(* IEC 61131-3 sources: RL_MAR/experiments/comparison/autoplc/results/deepseek-ai-DeepSeek-V3.2_20260508_111905/med_63, 1 file *)

(* ---- med_63_3.st ---- *)
FUNCTION MoveCarToExitGate : BOOL
VAR_INPUT
    SpaceNumber : INT;
END_VAR
VAR
    // Local variables if needed
END_VAR

(* This function simulates car movement to exit gate *)
(* In a real implementation, this would control physical actuators *)
(* For this example, we'll return TRUE immediately to indicate completion *)

MoveCarToExitGate := TRUE;
END_FUNCTION

FUNCTION_BLOCK Automated_Parking_Controller
VAR_INPUT
    EntryGateSensor : BOOL; (* Sensor input for entry gate *)
    ExitGateSensor : BOOL; (* Sensor input for exit gate *)
    CarDetected : BOOL; (* Sensor input for car detection *)
END_VAR
VAR_OUTPUT
    ParkingSpaceNumber : INT := 0; (* Allocated parking space number *)
    RetrievalInProgress : BOOL := FALSE; (* Flag for car retrieval in progress *)
END_VAR
VAR
    ParkingSpaces : ARRAY[1..100] OF BOOL; (* Parking space status: TRUE=Occupied, FALSE=Available *)
    i : INT; (* Loop counter *)
    EntryGateSensor_Prev : BOOL := FALSE; (* Previous state of entry gate sensor *)
    ExitGateSensor_Prev : BOOL := FALSE; (* Previous state of exit gate sensor *)
    CarDetected_Prev : BOOL := FALSE; (* Previous state of car detected sensor *)
    RetrievalSpaceNumber : INT := 0; (* Parking space number for retrieval *)
    MoveCarComplete : BOOL := FALSE; (* Flag for car movement completion *)
END_VAR

(* Initialization of parking spaces *)
FOR i := 1 TO 100 DO
    ParkingSpaces[i] := FALSE;
END_FOR;

(* Detect rising edge for EntryGateSensor *)
IF EntryGateSensor AND NOT EntryGateSensor_Prev THEN
    (* Entry gate management *)
    IF NOT RetrievalInProgress THEN
        (* Find first available parking space *)
        i := 1;
        WHILE i <= 100 DO
            IF NOT ParkingSpaces[i] THEN
                ParkingSpaces[i] := TRUE;
                ParkingSpaceNumber := i;
                EXIT;
            END_IF;
            i := i + 1;
        END_WHILE;
    END_IF;
END_IF;
EntryGateSensor_Prev := EntryGateSensor;

(* Detect rising edge for ExitGateSensor *)
IF ExitGateSensor AND NOT ExitGateSensor_Prev THEN
    (* Exit gate management *)
    IF ParkingSpaceNumber > 0 THEN
        ParkingSpaces[ParkingSpaceNumber] := FALSE;
        ParkingSpaceNumber := 0;
    END_IF;
END_IF;
ExitGateSensor_Prev := ExitGateSensor;

(* Detect rising edge for CarDetected *)
IF CarDetected AND NOT CarDetected_Prev THEN
    (* Car retrieval management *)
    IF NOT RetrievalInProgress AND ParkingSpaceNumber > 0 THEN
        RetrievalInProgress := TRUE;
        RetrievalSpaceNumber := ParkingSpaceNumber;
        MoveCarComplete := FALSE;
    END_IF;
END_IF;
CarDetected_Prev := CarDetected;

(* Execute retrieval process *)
IF RetrievalInProgress THEN
    IF NOT MoveCarComplete THEN
        MoveCarComplete := MoveCarToExitGate(SpaceNumber := RetrievalSpaceNumber);
    ELSE
        (* Car movement complete *)
        ParkingSpaces[RetrievalSpaceNumber] := FALSE;
        IF ParkingSpaceNumber = RetrievalSpaceNumber THEN
            ParkingSpaceNumber := 0;
        END_IF;
        RetrievalInProgress := FALSE;
        MoveCarComplete := FALSE;
    END_IF;
END_IF;
END_FUNCTION_BLOCK
